Fanuc KAREL source: kt00297.KL

PROGRAM KT00297
%STACKSIZE=65535
%PRIORITY=65535
%NOLOCKGROUP
VAR
R1 : REAL
I2 : INTEGER
OUT : BOOLEAN
BEGIN
R1=2.0
I2=3
-- UNSAFE_SOURCE_IR line 10: OUT = (R1 <> int_to_real(I2))
END KT00297
